{attribute 'GeneratedUsingTerminal: AT2050-0501-0017'}
{attribute addProperty BoxType "AT2050-0501-0017"}
{attribute addProperty Id "A_0088_AT2050_5501_0017_AT2050_5501AT2050_01D6DEDF80"}
{attribute addProperty CRC "869601335"}
{attribute addProperty Size "80"}
TYPE A_0056_AT2050_0501_0017_33D51037 EXTENDS AT2050_86175B41 :
STRUCT
	{attribute addProperty Name "A_0088_AT2050_5501_0017_AT2050_5501"}
	{attribute addProperty PreviousPort "A_0056(AT2050-0501-0017) : B"}
	A_0088_AT2050_5501_0017_AT2050_5501 : AT2050_01D6DEDF;
END_STRUCT
END_TYPE

(* stored: Version 1.2.0.0, ProductVersion 3.1.4024.9
   DUT A_0056_AT2050_0501_0017_33D51037: Id {768a6e42-3d71-487a-af32-2f4e03b24929} *)
